Fanuc KAREL source: kt00939.KL

-- PROVISIONAL review KL for V1013-1; original PC SHA256 d4183a2e916571f5acec4cbaf02552b5cff1145317a5d16880115e24f7cfd9c9
-- Incomplete behavior may be omitted. Consult companion uncertainty JSON. Do not deploy.
PROGRAM KT00939
%NOLOCKGROUP
VAR
  ENTRY : INTEGER
  PNAME : STRING[80]
  VNAME : STRING[80]
  STATUS : INTEGER
-- UNRESOLVED_DECL VALUE type=000101
BEGIN
  -- UNRESOLVED_PC offsets 5-12; opcodes 9C,23
  -- UNRESOLVED_PC offsets 17-25; opcodes 3F,75
  -- UNRESOLVED_PC offsets 30-43; opcodes 3F,75
  -- UNRESOLVED_PC offsets 48-92; opcodes 27,22,22,2A,22,2A,22,1C,22,AF
  -- UNRESOLVED_PC offsets 97-101; opcodes 7F
END KT00939
